(* Visualisation PLC_VISU
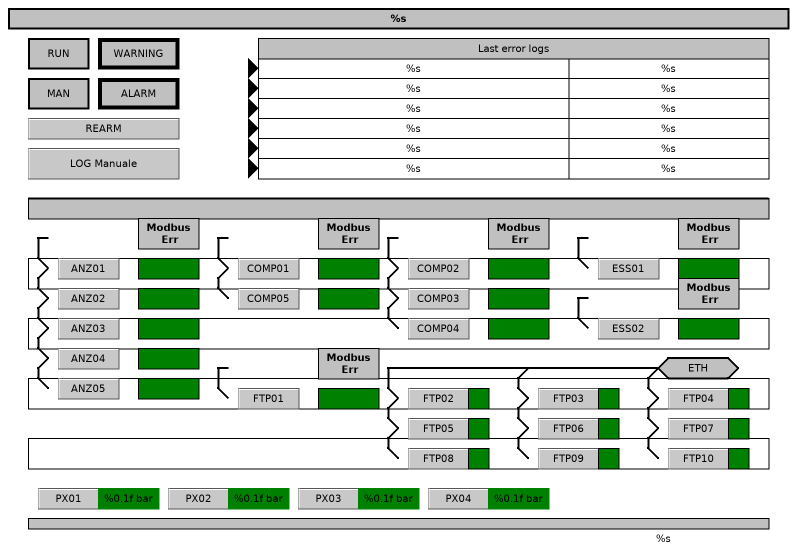
rectangle at (10,0)-(791,21): text "%s"; shows .Plant_NAME
rounded rectangle at (30,30)-(91,61): text "RUN"; alarm colour if NOT Mode_Manual; runs INTERN ASSIGN Mode_Manual:=(FALSE)
rounded rectangle at (30,70)-(91,101): text "MAN"; alarm colour if Mode_Manual; runs INTERN ASSIGN Mode_Manual:=(TRUE)
rectangle at (570,50)-(771,71): text "%s"; shows Sys.LastLogs_Msg[0]
polygon at (250,150)-(260,170): invisible if Sys.LastLogs_Idx<>0
rectangle at (570,70)-(771,91): text "%s"; shows Sys.LastLogs_Msg[1]
polygon at (250,50)-(260,70): invisible if Sys.LastLogs_Idx<>1
rectangle at (570,90)-(771,111): text "%s"; shows Sys.LastLogs_Msg[2]
polygon at (250,70)-(260,90): invisible if Sys.LastLogs_Idx<>2
rectangle at (570,110)-(771,131): text "%s"; shows Sys.LastLogs_Msg[3]
polygon at (250,90)-(260,110): invisible if Sys.LastLogs_Idx<>3
rectangle at (570,130)-(771,151): text "%s"; shows Sys.LastLogs_Msg[4]
polygon at (250,110)-(260,130): invisible if Sys.LastLogs_Idx<>4
rectangle at (570,150)-(771,171): text "%s"; shows Sys.LastLogs_Msg[5]
polygon at (250,130)-(260,150): invisible if Sys.LastLogs_Idx<>5
rectangle at (260,50)-(571,71): text "%s"; shows Sys.LastLogs_Dat[0]
rectangle at (260,70)-(571,91): text "%s"; shows Sys.LastLogs_Dat[1]
rectangle at (260,90)-(571,111): text "%s"; shows Sys.LastLogs_Dat[2]
rectangle at (260,110)-(571,131): text "%s"; shows Sys.LastLogs_Dat[3]
rectangle at (260,130)-(571,151): text "%s"; shows Sys.LastLogs_Dat[4]
rectangle at (260,150)-(571,171): text "%s"; shows Sys.LastLogs_Dat[5]
rectangle at (100,70)-(181,101): text "ALARM"; alarm colour if Sys.Alarm; runs INTERN ASSIGN Mode_Manual:=(FALSE)
rectangle at (100,30)-(181,61): text "WARNING"; alarm colour if Sys.Warning; runs INTERN ASSIGN Mode_Manual:=(TRUE)
button at (30,110)-(181,131): text "REARM"; runs INTERN ASSIGN Sys.Alarm:=(FALSE);INTERN ASSIGN Sys.Warning:=(FALSE)
button at (60,250)-(121,271): text "ANZ01"
rectangle at (260,30)-(771,51): text "Last error logs"
button at (60,280)-(121,301): text "ANZ02"
rectangle at (560,520)-(771,541): text "%s"; shows Sys.Time_LogString
rectangle at (140,210)-(201,241): text "Modbus / Err"
rectangle at (140,280)-(201,301): alarm colour if ANZ_MODBUS_CONNECTOR_INEPRO[2].fTimeout
button at (60,310)-(121,331): text "ANZ03"
rectangle at (140,310)-(201,331): alarm colour if ANZ_MODBUS_CONNECTOR_INEPRO[3].fTimeout
rectangle at (140,250)-(201,271): alarm colour if ANZ_MODBUS_CONNECTOR_INEPRO[1].fTimeout
button at (60,340)-(121,361): text "ANZ04"
rectangle at (140,340)-(201,361): alarm colour if ANZ_MODBUS_CONNECTOR_INEPRO[4].fTimeout
button at (60,370)-(121,391): text "ANZ05"
rectangle at (140,370)-(201,391): alarm colour if ANZ_MODBUS_CONNECTOR_INEPRO[5].fTimeout
button at (240,250)-(301,271): text "COMP01"
button at (240,280)-(301,301): text "COMP05"
rectangle at (320,250)-(381,271): alarm colour if .COMPRESSORE01.ErroreComuModBus
rectangle at (320,280)-(381,301): alarm colour if .COMPRESSORE05.ErroreComuModBus
rectangle at (320,210)-(381,241): text "Modbus / Err"
button at (410,250)-(471,271): text "COMP02"
button at (410,280)-(471,301): text "COMP03"
rectangle at (490,250)-(551,271): alarm colour if .COMPRESSORE02.ErroreComuModBus
rectangle at (490,280)-(551,301): alarm colour if .COMPRESSORE03.ErroreComuModBus
rectangle at (490,210)-(551,241): text "Modbus / Err"
button at (600,250)-(661,271): text "ESS01"
button at (600,310)-(661,331): text "ESS02"
rectangle at (680,250)-(741,271): alarm colour if ESSICATORE01.ErroreComuModBus
rectangle at (680,310)-(741,331): alarm colour if ESSICATORE02.ErroreComuModBus
rectangle at (680,210)-(741,241): text "Modbus / Err"
button at (240,380)-(301,401): text "FTP01"
rectangle at (320,380)-(381,401): alarm colour if .FPT01.ErroreComuModBus
rectangle at (320,340)-(381,371): text "Modbus / Err"
button at (410,310)-(471,331): text "COMP04"
rectangle at (490,310)-(551,331): alarm colour if .COMPRESSORE04.ErroreComuModBus
button at (40,480)-(101,501): text "PX01"
rectangle at (100,480)-(161,501): text "%0.1f bar"; shows INT_TO_REAL(.PX01.ValoreScalato)/10
button at (170,480)-(231,501): text "PX02"
rectangle at (230,480)-(291,501): text "%0.1f bar"; shows INT_TO_REAL(.PX02.ValoreScalato)/10
button at (300,480)-(361,501): text "PX03"
rectangle at (360,480)-(421,501): text "%0.1f bar"; shows INT_TO_REAL(.PX03.ValoreScalato)/10
button at (430,480)-(491,501): text "PX04"
rectangle at (490,480)-(551,501): text "%0.1f bar"; shows INT_TO_REAL(.PX04.ValoreScalato)/10
button at (30,140)-(181,171): text "LOG Manuale"; taps PLC_PRG.HMI_AggiornaLog
button at (410,380)-(471,401): text "FTP02"
polygon at (660,350)-(740,370): text "ETH"
rectangle at (470,380)-(491,401): alarm colour if .FPT02.ErroreComuModBus
button at (540,380)-(601,401): text "FTP03"
rectangle at (600,380)-(621,401): alarm colour if .FPT03.ErroreComuModBus
button at (670,380)-(731,401): text "FTP04"
rectangle at (730,380)-(751,401): alarm colour if .FPT04.ErroreComuModBus
button at (410,410)-(471,431): text "FTP05"
rectangle at (470,410)-(491,431): alarm colour if .FPT05.ErroreComuModBus
button at (540,410)-(601,431): text "FTP06"
rectangle at (600,410)-(621,431): alarm colour if .FPT06.ErroreComuModBus
button at (670,410)-(731,431): text "FTP07"
rectangle at (730,410)-(751,431): alarm colour if .FPT07.ErroreComuModBus
button at (670,440)-(731,461): text "FTP10"
rectangle at (730,440)-(751,461): alarm colour if .FPT10.ErroreComuModBus
button at (540,440)-(601,461): text "FTP09"
rectangle at (600,440)-(621,461): alarm colour if .FPT09.ErroreComuModBus
button at (410,440)-(471,461): text "FTP08"
rectangle at (470,440)-(491,461): alarm colour if .FPT08.ErroreComuModBus
rectangle at (680,270)-(741,301): text "Modbus / Err"
29 more shapes without text or variables
28 elements of other kinds (tables, trends, ...) not read
*)

(* Visualisation PLC_VISU_COMP
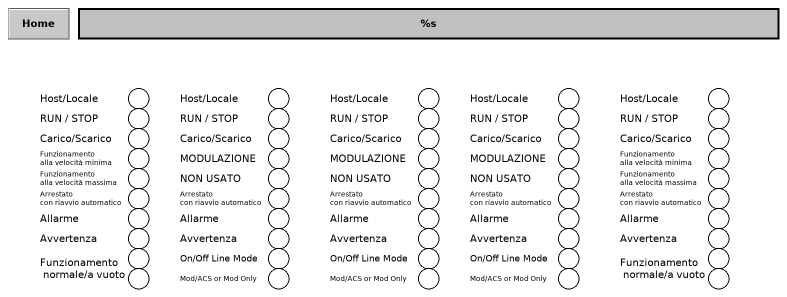
button at (10,10)-(71,41): text "Home"; opens PLC_VISU
rectangle at (80,10)-(781,41): text "%s"; shows .Plant_NAME
ellipse at (130,90)-(151,111): alarm colour if .COMPRESSORE01.StatusControl[0]
ellipse at (130,110)-(151,131): alarm colour if .COMPRESSORE01.StatusControl[1]
ellipse at (130,130)-(151,151): alarm colour if .COMPRESSORE01.StatusControl[2]
ellipse at (130,150)-(151,171): alarm colour if .COMPRESSORE01.StatusControl[3]
ellipse at (130,170)-(151,191): alarm colour if .COMPRESSORE01.StatusControl[4]
ellipse at (130,190)-(151,211): alarm colour if .COMPRESSORE01.StatusControl[5]
ellipse at (130,210)-(151,231): alarm colour if .COMPRESSORE01.StatusControl[6]
ellipse at (130,230)-(151,251): alarm colour if .COMPRESSORE01.StatusControl[7]
ellipse at (130,250)-(151,271): alarm colour if .COMPRESSORE01.StatusControl[8]
ellipse at (130,270)-(151,291): alarm colour if .COMPRESSORE01.StatusControl[9]
rectangle at (40,90)-(131,111): text "Host/Locale"
rectangle at (40,110)-(131,131): text "RUN / STOP"
rectangle at (40,130)-(131,151): text "Carico/Scarico"
rectangle at (40,140)-(131,181): text "Funzionamento / alla velocità minima"
rectangle at (40,170)-(131,191): text "Funzionamento / alla velocità massima"
rectangle at (40,190)-(131,211): text "Arrestato / con riavvio automatico"
rectangle at (40,210)-(131,231): text "Allarme"
rectangle at (40,230)-(131,251): text "Avvertenza"
rectangle at (40,250)-(131,291): text "Funzionamento / normale/a vuoto"
ellipse at (710,90)-(731,111): alarm colour if .COMPRESSORE05.StatusControl[0]
ellipse at (710,110)-(731,131): alarm colour if .COMPRESSORE05.StatusControl[1]
ellipse at (710,130)-(731,151): alarm colour if .COMPRESSORE05.StatusControl[2]
ellipse at (710,150)-(731,171): alarm colour if .COMPRESSORE05.StatusControl[3]
ellipse at (710,170)-(731,191): alarm colour if .COMPRESSORE05.StatusControl[4]
ellipse at (710,190)-(731,211): alarm colour if .COMPRESSORE05.StatusControl[5]
ellipse at (710,210)-(731,231): alarm colour if .COMPRESSORE05.StatusControl[6]
ellipse at (710,230)-(731,251): alarm colour if .COMPRESSORE05.StatusControl[7]
ellipse at (710,250)-(731,271): alarm colour if .COMPRESSORE05.StatusControl[8]
ellipse at (710,270)-(731,291): alarm colour if .COMPRESSORE05.StatusControl[9]
rectangle at (620,90)-(711,111): text "Host/Locale"
rectangle at (620,110)-(711,131): text "RUN / STOP"
rectangle at (620,130)-(711,151): text "Carico/Scarico"
rectangle at (620,140)-(711,181): text "Funzionamento / alla velocità minima"
rectangle at (620,170)-(711,191): text "Funzionamento / alla velocità massima"
rectangle at (620,190)-(711,211): text "Arrestato / con riavvio automatico"
rectangle at (620,210)-(711,231): text "Allarme"
rectangle at (620,230)-(711,251): text "Avvertenza"
rectangle at (620,250)-(711,291): text "Funzionamento / normale/a vuoto"
ellipse at (270,90)-(291,111): alarm colour if .COMPRESSORE02.StatusControl[0]
ellipse at (270,110)-(291,131): alarm colour if .COMPRESSORE02.StatusControl[1]
ellipse at (270,130)-(291,151): alarm colour if .COMPRESSORE02.StatusControl[2]
ellipse at (270,150)-(291,171): alarm colour if .COMPRESSORE02.StatusControl[3]
ellipse at (270,170)-(291,191): alarm colour if .COMPRESSORE02.StatusControl[4]
ellipse at (270,190)-(291,211): alarm colour if .COMPRESSORE02.StatusControl[5]
ellipse at (270,210)-(291,231): alarm colour if .COMPRESSORE02.StatusControl[6]
ellipse at (270,230)-(291,251): alarm colour if .COMPRESSORE02.StatusControl[7]
ellipse at (270,250)-(291,271): alarm colour if .COMPRESSORE02.StatusControl[8]
ellipse at (270,270)-(291,291): alarm colour if .COMPRESSORE02.StatusControl[9]
rectangle at (180,90)-(271,111): text "Host/Locale"
rectangle at (180,110)-(271,131): text "RUN / STOP"
rectangle at (180,130)-(271,151): text "Carico/Scarico"
rectangle at (180,140)-(271,181): text "MODULAZIONE"
rectangle at (180,170)-(271,191): text "NON USATO"
rectangle at (180,190)-(271,211): text "Arrestato / con riavvio automatico"
rectangle at (180,210)-(271,231): text "Allarme"
rectangle at (180,230)-(271,251): text "Avvertenza"
rectangle at (180,250)-(271,271): text "On/Off Line Mode"
rectangle at (180,270)-(271,291): text "Mod/ACS or Mod Only"
ellipse at (420,90)-(441,111): alarm colour if .COMPRESSORE03.StatusControl[0]
ellipse at (420,110)-(441,131): alarm colour if .COMPRESSORE03.StatusControl[1]
ellipse at (420,130)-(441,151): alarm colour if .COMPRESSORE03.StatusControl[2]
ellipse at (420,150)-(441,171): alarm colour if .COMPRESSORE03.StatusControl[3]
ellipse at (420,170)-(441,191): alarm colour if .COMPRESSORE03.StatusControl[4]
ellipse at (420,190)-(441,211): alarm colour if .COMPRESSORE03.StatusControl[5]
ellipse at (420,210)-(441,231): alarm colour if .COMPRESSORE03.StatusControl[6]
ellipse at (420,230)-(441,251): alarm colour if .COMPRESSORE03.StatusControl[7]
ellipse at (420,250)-(441,271): alarm colour if .COMPRESSORE03.StatusControl[8]
ellipse at (420,270)-(441,291): alarm colour if .COMPRESSORE03.StatusControl[9]
rectangle at (330,90)-(421,111): text "Host/Locale"
rectangle at (330,110)-(421,131): text "RUN / STOP"
rectangle at (330,130)-(421,151): text "Carico/Scarico"
rectangle at (330,140)-(421,181): text "MODULAZIONE"
rectangle at (330,170)-(421,191): text "NON USATO"
rectangle at (330,190)-(421,211): text "Arrestato / con riavvio automatico"
rectangle at (330,210)-(421,231): text "Allarme"
rectangle at (330,230)-(421,251): text "Avvertenza"
rectangle at (330,250)-(421,271): text "On/Off Line Mode"
rectangle at (330,270)-(421,291): text "Mod/ACS or Mod Only"
ellipse at (560,90)-(581,111): alarm colour if .COMPRESSORE04.StatusControl[0]
ellipse at (560,110)-(581,131): alarm colour if .COMPRESSORE04.StatusControl[1]
ellipse at (560,130)-(581,151): alarm colour if .COMPRESSORE04.StatusControl[2]
ellipse at (560,150)-(581,171): alarm colour if .COMPRESSORE04.StatusControl[3]
ellipse at (560,170)-(581,191): alarm colour if .COMPRESSORE04.StatusControl[4]
ellipse at (560,190)-(581,211): alarm colour if .COMPRESSORE04.StatusControl[5]
ellipse at (560,210)-(581,231): alarm colour if .COMPRESSORE04.StatusControl[6]
ellipse at (560,230)-(581,251): alarm colour if .COMPRESSORE04.StatusControl[7]
ellipse at (560,250)-(581,271): alarm colour if .COMPRESSORE04.StatusControl[8]
ellipse at (560,270)-(581,291): alarm colour if .COMPRESSORE04.StatusControl[9]
rectangle at (470,90)-(561,111): text "Host/Locale"
rectangle at (470,110)-(561,131): text "RUN / STOP"
rectangle at (470,130)-(561,151): text "Carico/Scarico"
rectangle at (470,140)-(561,181): text "MODULAZIONE"
rectangle at (470,170)-(561,191): text "NON USATO"
rectangle at (470,190)-(561,211): text "Arrestato / con riavvio automatico"
rectangle at (470,210)-(561,231): text "Allarme"
rectangle at (470,230)-(561,251): text "Avvertenza"
rectangle at (470,250)-(561,271): text "On/Off Line Mode"
rectangle at (470,270)-(561,291): text "Mod/ACS or Mod Only"
5 elements of other kinds (tables, trends, ...) not read
*)

(* Visualisation PLC_VISU_FTP
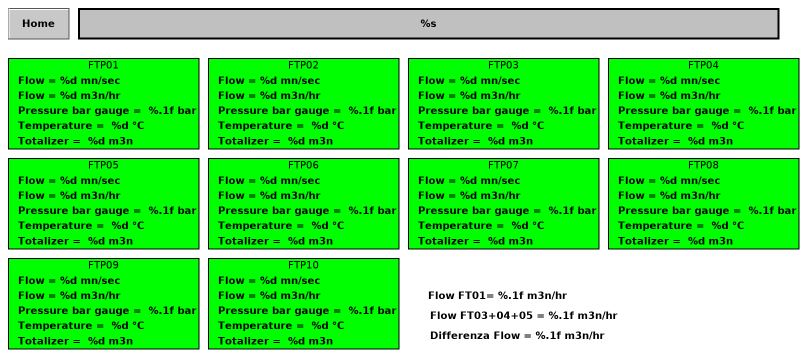
button at (10,10)-(71,41): text "Home"; opens PLC_VISU
rectangle at (80,10)-(781,41): text "%s"; shows .Plant_NAME
group at (210,60)-(401,151)
  rectangle at (0,0)-(191,91): text "FTP02"
  rectangle at (8,15)-(174,30): text "Flow = %d mn/sec"; shows .FPT02.Parametro16
  rectangle at (8,30)-(182,45): text "Flow = %d m3n/hr"; shows .FPT02.Parametro18
  rectangle at (8,45)-(182,60): text "Pressure bar gauge =  %.1f bar"; shows DWORD_TO_REAL(.FPT02.Parametro32)/10
  rectangle at (8,60)-(182,75): text "Temperature =  %d °C"; shows .FPT02.Parametro64
  rectangle at (8,75)-(182,91): text "Totalizer =  %d m3n"; shows .FPT02.Parametro128
group at (410,60)-(601,151)
  rectangle at (0,0)-(191,91): text "FTP03"
  rectangle at (8,15)-(174,30): text "Flow = %d mn/sec"; shows .FPT03.Parametro16
  rectangle at (8,30)-(182,45): text "Flow = %d m3n/hr"; shows .FPT03.Parametro18
  rectangle at (8,45)-(182,60): text "Pressure bar gauge =  %.1f bar"; shows DWORD_TO_REAL(.FPT03.Parametro32)/10
  rectangle at (8,60)-(182,75): text "Temperature =  %d °C"; shows .FPT03.Parametro64
  rectangle at (8,75)-(182,91): text "Totalizer =  %d m3n"; shows .FPT03.Parametro128
group at (610,60)-(801,151)
  rectangle at (0,0)-(191,91): text "FTP04"
  rectangle at (8,15)-(174,30): text "Flow = %d mn/sec"; shows .FPT04.Parametro16
  rectangle at (8,30)-(182,45): text "Flow = %d m3n/hr"; shows .FPT04.Parametro18
  rectangle at (8,45)-(182,60): text "Pressure bar gauge =  %.1f bar"; shows DWORD_TO_REAL(.FPT04.Parametro32)/10
  rectangle at (8,60)-(182,75): text "Temperature =  %d °C"; shows .FPT04.Parametro64
  rectangle at (8,75)-(182,91): text "Totalizer =  %d m3n"; shows .FPT04.Parametro128
group at (10,160)-(201,251)
  rectangle at (0,0)-(191,91): text "FTP05"
  rectangle at (8,15)-(174,30): text "Flow = %d mn/sec"; shows .FPT05.Parametro16
  rectangle at (8,30)-(182,45): text "Flow = %d m3n/hr"; shows .FPT05.Parametro18
  rectangle at (8,45)-(182,60): text "Pressure bar gauge =  %.1f bar"; shows DWORD_TO_REAL(.FPT05.Parametro32)/10
  rectangle at (8,60)-(182,75): text "Temperature =  %d °C"; shows .FPT05.Parametro64
  rectangle at (8,75)-(182,91): text "Totalizer =  %d m3n"; shows .FPT05.Parametro128
group at (210,160)-(401,251)
  rectangle at (0,0)-(191,91): text "FTP06"
  rectangle at (8,15)-(174,30): text "Flow = %d mn/sec"; shows .FPT06.Parametro16
  rectangle at (8,30)-(182,45): text "Flow = %d m3n/hr"; shows .FPT06.Parametro18
  rectangle at (8,45)-(182,60): text "Pressure bar gauge =  %.1f bar"; shows DWORD_TO_REAL(.FPT06.Parametro32)/10
  rectangle at (8,60)-(182,75): text "Temperature =  %d °C"; shows .FPT06.Parametro64
  rectangle at (8,75)-(182,91): text "Totalizer =  %d m3n"; shows .FPT06.Parametro128
group at (410,160)-(601,251)
  rectangle at (0,0)-(191,91): text "FTP07"
  rectangle at (8,15)-(174,30): text "Flow = %d mn/sec"; shows .FPT07.Parametro16
  rectangle at (8,30)-(182,45): text "Flow = %d m3n/hr"; shows .FPT07.Parametro18
  rectangle at (8,45)-(182,60): text "Pressure bar gauge =  %.1f bar"; shows DWORD_TO_REAL(.FPT07.Parametro32)/10
  rectangle at (8,60)-(182,75): text "Temperature =  %d °C"; shows .FPT07.Parametro64
  rectangle at (8,75)-(182,91): text "Totalizer =  %d m3n"; shows .FPT07.Parametro128
group at (610,160)-(801,251)
  rectangle at (0,0)-(191,91): text "FTP08"
  rectangle at (8,15)-(174,30): text "Flow = %d mn/sec"; shows .FPT08.Parametro16
  rectangle at (8,30)-(182,45): text "Flow = %d m3n/hr"; shows .FPT08.Parametro18
  rectangle at (8,45)-(182,60): text "Pressure bar gauge =  %.1f bar"; shows DWORD_TO_REAL(.FPT08.Parametro32)/10
  rectangle at (8,60)-(182,75): text "Temperature =  %d °C"; shows .FPT08.Parametro64
  rectangle at (8,75)-(182,91): text "Totalizer =  %d m3n"; shows .FPT08.Parametro128
rectangle at (428,290)-(701,305): text "Flow FT01= %.1f m3n/hr"; shows DWORD_TO_REAL(.FPT01.Parametro17)
rectangle at (430,310)-(681,325): text "Flow FT03+04+05 = %.1f m3n/hr"; shows DWORD_TO_REAL((.FPT03.Parametro18+.FPT04.Parametro18+.FPT05.Parametro18)/10)
rectangle at (430,330)-(701,345): text "Differenza Flow = %.1f m3n/hr"; shows DWORD_TO_REAL(.FPT01.Parametro17-(.FPT03.Parametro18+.FPT04.Parametro18+.FPT05.Parametro18)/10)
group at (10,60)-(201,151)
  rectangle at (0,0)-(191,91): text "FTP01"
  rectangle at (8,15)-(174,30): text "Flow = %d mn/sec"; shows .FPT01.Parametro16
  rectangle at (8,30)-(182,45): text "Flow = %d m3n/hr"; shows .FPT01.Parametro17
  rectangle at (8,45)-(182,60): text "Pressure bar gauge =  %.1f bar"; shows .FPT01.PressioneCalcolata
  rectangle at (8,60)-(182,75): text "Temperature =  %d °C"; shows .FPT01.Parametro64
  rectangle at (8,75)-(182,91): text "Totalizer =  %d m3n"; shows .FPT01.Parametro128
group at (10,260)-(201,351)
  rectangle at (0,0)-(191,91): text "FTP09"
  rectangle at (8,15)-(174,30): text "Flow = %d mn/sec"; shows .FPT09.Parametro16
  rectangle at (8,30)-(182,45): text "Flow = %d m3n/hr"; shows .FPT09.Parametro18
  rectangle at (8,45)-(182,60): text "Pressure bar gauge =  %.1f bar"; shows DWORD_TO_REAL(.FPT09.Parametro32)/10
  rectangle at (8,60)-(182,75): text "Temperature =  %d °C"; shows .FPT09.Parametro64
  rectangle at (8,75)-(182,91): text "Totalizer =  %d m3n"; shows .FPT09.Parametro128
group at (210,260)-(401,351)
  rectangle at (0,0)-(191,91): text "FTP10"
  rectangle at (8,15)-(174,30): text "Flow = %d mn/sec"; shows .FPT10.Parametro16
  rectangle at (8,30)-(182,45): text "Flow = %d m3n/hr"; shows .FPT10.Parametro18
  rectangle at (8,45)-(182,60): text "Pressure bar gauge =  %.1f bar"; shows DWORD_TO_REAL(.FPT10.Parametro32)/10
  rectangle at (8,60)-(182,75): text "Temperature =  %d °C"; shows .FPT10.Parametro64
  rectangle at (8,75)-(182,91): text "Totalizer =  %d m3n"; shows .FPT10.Parametro128
*)

(* Visualisation PLC_VISU_raw_data
rectangle at (10,0)-(871,21): text "%s"; shows .Plant_NAME
3 elements of other kinds (tables, trends, ...) not read
*)

(* Visualisation PLC_VISU_raw_data_BIS
rectangle at (10,0)-(791,21): text "%s"; shows .Plant_NAME
3 elements of other kinds (tables, trends, ...) not read
*)

(* Visualisation PLC_VISU_raw_data_tris
rectangle at (10,0)-(791,21): text "%s"; shows .Plant_NAME
2 elements of other kinds (tables, trends, ...) not read
*)
